PROGRAM CraneSimulation
VAR
	fTime : LREAL; 	
	fPositionAutoMode : LREAL; 
	fInitialPosition : LREAL; 
	fInitialVelocity : LREAL;  
	bPistonMaxNewValue : BOOL;
	fPressureEng : REAL;
	fFlowEng : REAL;
	fPressureBar : LREAL := 60;
	fFlowLmin : LREAL := 20;
	fBoomAngleRad : LREAL;
	fBoomAnimation : LREAL;
	fbModeSelector : FB_ModeSelector;
	fbStatus : FB_Status;
	fbSimulationTime : FB_SimulationTime;
	fbPositionSimulator : FB_PositionSimulator;
END_VAR

// Status
fbStatus(
bPowerOn := HMI.bPowerOn,
bFault := FALSE,
bStart:= HMI.bStart,
bStop := HMI.bStop,
bRunning := HMI.bRunning,
eStatus => HMI.eStatus
);

// Mode Selector
fbModeSelector(bControlBox := FALSE);

// Simulation Time
fbSimulationTime(
eMode := HMI.eMode,
eStatus := HMI.eStatus,
stParam := Parameters.stParam,
fTime => HMI.fSimulationTime
);

// Position Simulation and Animation
IF  HMI.eStatus = E_Status.Ready OR HMI.eStatus = E_Status.Starting OR HMI.eStatus = E_Status.Running THEN
	fbPositionSimulator(
		eMode := HMI.eMode,
		stParam := Parameters.stParam,
		fTime := HMI.fSimulationTime,
		fPositionReference := HMI.fManualCylinderPositionReference,
		fVelocityReference := HMI.fCylinderVelocityReference,
		fInitialVelocity := 0.0,
		fInitialPosition := 0.0,
		bRunning => HMI.bRunning,
		sPistonEndStopMessages => HMI.sPistonEndStopMessages,
		fPositionRestricted => HMI.fCylinderPosition,
		stBoomAnimation => HMI.stBoomAnimation,
		stPistonAnimation => HMI.stPistonAnimation,
		fBoomAngleDeg =>  HMI.fBoomAngleDeg
	);
END_IF

F_UpdateParametersByReference( 
	bSetNewValue := bPistonMaxNewValue,
	fMaxPistonStroke := HMI.fMaxPistonPosition,
	paramCylinderPiston := Parameters.stParam.stPistonRange
);

END_PROGRAM

(* stored: Version 1.1.0.1, ProductVersion 3.1.4024.10
   POU CraneSimulation: Id {c255987f-7a58-4573-9ac9-545c12e8d4a5}, SpecialFunc None *)
